FUNCTION_BLOCK NEGATIVEEdge
	VAR_INPUT
		IN         : BOOL;
		INprevious : BOOL;
	END_VAR
	VAR_OUTPUT
		OUT : BOOL;
	END_VAR
BEGIN
	OUT := BOOL_TO_DINT(IN) < BOOL_TO_DINT(INprevious);
END_FUNCTION_BLOCK